FUNCTION GetBuild : UINT
VAR_INPUT
END_VAR
VAR
END_VAR

GetBuild := Version.Build;

END_FUNCTION

(* stored: Version 1.1.0.1, ProductVersion 3.1.4024.0
   POU GetBuild: Id {db5f19de-3a4e-4ca1-86fc-ec1c67798d00}, SpecialFunc None *)
